KUKA KRL program: FORCE_NEG_Y2.src, FORCE_NEG_Y2.dat

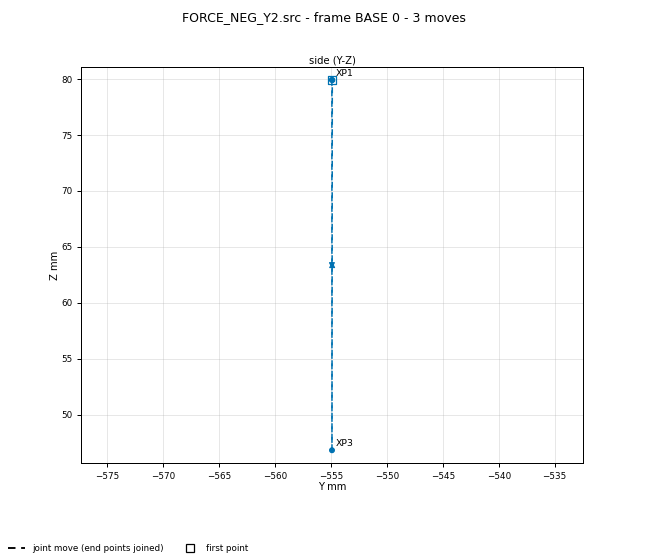
[picture p0: tool path of FORCE_NEG_Y2.src in frame BASE 0, 3 of 3 moves have a stored position in this frame; points joined in program order, loops and branches not executed]
--- FORCE_NEG_Y2.src ---
&ACCESS RVO
&REL 59
&PARAM TEMPLATE = C:\KRC\Roboter\Template\vorgabe
&PARAM EDITMASK = *
DEF FORCE_NEG_Y2( )
DECL BOOL TEMP, HEMP, SEMP
DECL INT md_int[16]
DECL REAL md_real[16]
DECL INT n, result

;FOLD INI
  ;FOLD BASISTECH INI
    GLOBAL INTERRUPT DECL 3 WHEN $STOPMESS==TRUE DO IR_STOPM ( )
    INTERRUPT ON 3
    BAS (#INITMOV,0 )
  ;ENDFOLD (BASISTECH INI)
  ;FOLD USER INI
    ;Make your modifications here

  ;ENDFOLD (USER INI)
;ENDFOLD (INI)

$STIFFNESS.STRATEGY=10
$STIFFNESS.COMMIT=TRUE
$OV_PRO=75
$ORI_TYPE=#CONSTANT
$TOOL=TOOL_DATA[5]
$VEL.CP=1.0
$VEL.ORI1=150
$VEL.ORI2=100
$ACC.CP=1.7
$ACC.ORI1=80
$ACC.ORI2=80


;FOLD PTP P1 Vel=100 % PDAT1 Tool[5]:Pneumatic_gripper_probe Base[0];%{PE}%R 5.6.11,%MKUKATPBASIS,%CMOVE,%VPTP,%P 1:PTP, 2:P1, 3:, 5:100, 7:PDAT1
$BWDSTART=FALSE
PDAT_ACT=PPDAT1
FDAT_ACT=FP1
BAS(#PTP_PARAMS,100)
PTP XP1
;ENDFOLD

;FOLD PTP P3 Vel=100 % PDAT3 Tool[5]:Pneumatic_gripper_probe Base[0];%{PE}%R 5.6.11,%MKUKATPBASIS,%CMOVE,%VPTP,%P 1:PTP, 2:P3, 3:, 5:100, 7:PDAT3
$BWDSTART=FALSE
PDAT_ACT=PPDAT3
FDAT_ACT=FP3
BAS(#PTP_PARAMS,100)
PTP XP3
;ENDFOLD


TEMP=TRIGY()

SEMP=SETSTIFF("Y",1.0)

HEMP=SETFORCE("Y",5.0)

$OV_PRO=10
LIN_REL{Y -5}

HALT



;FOR n=1 TO 16
;md_int[n]=0
;md_real[n]=0
;ENDFOR
;md_real[1]=0.05

;result=MD_CMD("PAPAS","TRIGBYCONTACT",md_int[],md_real[])

$STIFFNESS.STRATEGY=10
$STIFFNESS.COMMIT=TRUE
$OV_PRO=50


;FOLD PTP P2 Vel=100 % PDAT2 Tool[5]:Pneumatic_gripper_probe Base[0];%{PE}%R 5.6.11,%MKUKATPBASIS,%CMOVE,%VPTP,%P 1:PTP, 2:P2, 3:, 5:100, 7:PDAT2
$BWDSTART=FALSE
PDAT_ACT=PPDAT2
FDAT_ACT=FP2
BAS(#PTP_PARAMS,100)
PTP XP2
;ENDFOLD

END

--- FORCE_NEG_Y2.dat ---
&ACCESS RVO
&REL 59
&PARAM TEMPLATE = C:\KRC\Roboter\Template\vorgabe
&PARAM EDITMASK = *
DEFDAT  FORCE_NEG_Y2
;FOLD EXTERNAL DECLARATIONS;%{PE}%MKUKATPBASIS,%CEXT,%VCOMMON,%P
;FOLD BASISTECH EXT;%{PE}%MKUKATPBASIS,%CEXT,%VEXT,%P
EXT  BAS (BAS_COMMAND  :IN,REAL  :IN )
DECL INT SUCCESS
;ENDFOLD (BASISTECH EXT)
;FOLD USER EXT;%{E}%MKUKATPUSER,%CEXT,%VEXT,%P
;Make here your modifications

;ENDFOLD (USER EXT)
;ENDFOLD (EXTERNAL DECLARATIONS)
DECL BASIS_SUGG_T LAST_BASIS={POINT1[] "P3                      ",POINT2[] "P3                      ",CP_PARAMS[] "CPDAT0                  ",PTP_PARAMS[] "PDAT3                   ",CONT[] "                        ",CP_VEL[] "2.0                     ",PTP_VEL[] "100                     ",SYNC_PARAMS[] "SYNCDAT                 ",SPL_NAME[] "S0                      "}
DECL E6POS XP1={X 14.99335,Y -554.926819,Z 79.9336777,A -0.000569114287,B 0.00111991004,C -179.987595,S 1,T 44,E1 -6.86645508E-05,E2 0.0,E3 0.0,E4 0.0,E5 0.0,E6 0.0}
DECL FDAT FP1={TOOL_NO 5,BASE_NO 0,IPO_FRAME #BASE,POINT2[] " ",TQ_STATE FALSE}
DECL PDAT PPDAT1={VEL 100.0,ACC 100.0,APO_DIST 100.0,APO_MODE #CPTP}
DECL E6POS XP2={X 14.9922504,Y -554.888184,Z 79.9055023,A 0.00448764907,B 0.00187605806,C -179.979904,S 1,T 44,E1 -0.000360488892,E2 0.0,E3 0.0,E4 0.0,E5 0.0,E6 0.0}
DECL FDAT FP2={TOOL_NO 5,BASE_NO 0,IPO_FRAME #BASE,POINT2[] " ",TQ_STATE FALSE}
DECL PDAT PPDAT2={VEL 100.0,ACC 100.0,APO_DIST 100.0,APO_MODE #CPTP}
DECL E6POS XP3={X 14.9937696,Y -554.917908,Z 46.807209,A -0.000219844602,B 0.00128428801,C -179.986694,S 1,T 44,E1 -6.86645508E-05,E2 0.0,E3 0.0,E4 0.0,E5 0.0,E6 0.0}
DECL FDAT FP3={TOOL_NO 5,BASE_NO 0,IPO_FRAME #BASE,POINT2[] " ",TQ_STATE FALSE}
DECL PDAT PPDAT3={VEL 100.0,ACC 100.0,APO_DIST 100.0,APO_MODE #CPTP}
ENDDAT
